ORGANIZATION_BLOCK MAIN:OB1
TITLE= ==========================================
//  初始化与急停复位
//  ==========================================
BEGIN
Network 1 //  首次扫描初始化（清零状态与输出）
LD     SM0.1  // 读取 首次扫描(SM0.1)
MOVB   0, VB100  // 开机顺控状态清零
MOVB   0, VB101  // 关机顺控状态清零
R      Q0.0, 8  // 复位输出 Q0.0~Q0.7
R      Q1.0, 1  // 复位 直流电源(Q1.0)，数量=1
R      M0.0, 2  // 复位 M0.0~M0.1（泵使能）

Network 2 //  急停处理（I0.3）
LD     I0.3  // 读取 急停(I0.3)
MOVB   0, VB100  // 开机顺控状态清零
MOVB   0, VB101  // 关机顺控状态清零
R      Q0.0, 8  // 复位输出 Q0.0~Q0.7
R      Q1.0, 1  // 复位 直流电源(Q1.0)，数量=1
R      M0.0, 2  // 复位 M0.0~M0.1（泵使能）

// ==========================================
// 开机关机触发
// ==========================================
Network 3 //  开机触发（I0.1）
LD     I0.1  // 读取 开机按钮(I0.1)
AN     I0.3  // 与非 急停(I0.3)
AB=    VB100, 0  // 判断 开机顺控状态(VB100) = 0
AB=    VB101, 0  // 判断 关机顺控状态(VB101) = 0
MOVB   10, VB100  // 开机进入步骤10（补水）

Network 4 //  关机触发（I0.2）
LD     I0.2  // 读取 关机按钮(I0.2)
AN     I0.3  // 与非 急停(I0.3)
MOVB   0, VB100  // 开机顺控状态清零
MOVB   10, VB101  // 关机进入步骤10（立即停）

// ==========================================
// AE08 模拟量采集 (8路 4-20mA)
// 说明：按 S7-200 SMART 的固定映射惯例，首个右侧信号模块的模拟量起始通常为 AIW16。
// 若你的系统块里显示的起始地址不同，只需改这里的 AIWxx。
// ==========================================
Network 5 //  AE08 CH0 采集：压力 -> VW1000
LD     SM0.0  // 读取 Always_On(SM0.0)
MOVW   AIW16, VW1000  // 采集模拟量到 压力原始值(VW1000)

Network 6 //  AE08 CH1 采集：阳极液位 -> VW1002
LD     SM0.0  // 读取 Always_On(SM0.0)
MOVW   AIW18, VW1002  // 采集模拟量到 阳极液位原始值(VW1002)

Network 7 //  AE08 CH2 采集：阴极液位 -> VW1004
LD     SM0.0  // 读取 Always_On(SM0.0)
MOVW   AIW20, VW1004  // 采集模拟量到 阴极液位原始值(VW1004)

Network 8 //  AE08 CH3 预留 -> VW1010
LD     SM0.0  // 读取 Always_On(SM0.0)
MOVW   AIW22, VW1010  // 采集模拟量到 VW1010

Network 9 //  AE08 CH4 预留 -> VW1012
LD     SM0.0  // 读取 Always_On(SM0.0)
MOVW   AIW24, VW1012  // 采集模拟量到 VW1012

Network 10 //  AE08 CH5 预留 -> VW1014
LD     SM0.0  // 读取 Always_On(SM0.0)
MOVW   AIW26, VW1014  // 采集模拟量到 VW1014

Network 11 //  AE08 CH6 预留 -> VW1016
LD     SM0.0  // 读取 Always_On(SM0.0)
MOVW   AIW28, VW1016  // 采集模拟量到 VW1016

Network 12 //  AE08 CH7 预留 -> VW1018
LD     SM0.0  // 读取 Always_On(SM0.0)
MOVW   AIW30, VW1018  // 采集模拟量到 VW1018

// ==========================================
// 开机顺控状态机 (VB100)
// ==========================================
Network 13 //  开机步骤10：开制水+开补水阀
LD     SM0.0  // 读取 Always_On(SM0.0)
AB=    VB100, 10  // 判断 开机顺控状态(VB100) = 10
S      Q0.7, 1  // 置位 制水机(Q0.7)
S      Q0.2, 1  // 置位 阳极补水阀(Q0.2)
S      Q0.3, 1  // 置位 阴极补水阀(Q0.3)

Network 14 //  开机步骤10：阳极液位达标关阳极补水
LD     SM0.0  // 读取 Always_On(SM0.0)
AB=    VB100, 10  // 判断 开机顺控状态(VB100) = 10
AW>=   VW1002, 100  // 模拟量阈值比较（达到则进入下一步）
R      Q0.2, 1  // 复位 阳极补水阀(Q0.2)，数量=1

Network 15 //  开机步骤10：阴极液位达标关阴极补水
LD     SM0.0  // 读取 Always_On(SM0.0)
AB=    VB100, 10  // 判断 开机顺控状态(VB100) = 10
AW>=   VW1004, 100  // 模拟量阈值比较（达到则进入下一步）
R      Q0.3, 1  // 复位 阴极补水阀(Q0.3)，数量=1

Network 16 //  开机步骤10：两路补水阀都关 -> 进入步骤20
LD     SM0.0  // 读取 Always_On(SM0.0)
AB=    VB100, 10  // 判断 开机顺控状态(VB100) = 10
AN     Q0.2  // 与非 阳极补水阀(Q0.2)
AN     Q0.3  // 与非 阴极补水阀(Q0.3)
MOVB   20, VB100  // 开机进入步骤20（空压机）

Network 17 //  开机步骤20：启动空压机并计时3秒
LD     SM0.0  // 读取 Always_On(SM0.0)
AB=    VB100, 20  // 判断 开机顺控状态(VB100) = 20
S      Q0.6, 1  // 置位 空压机(Q0.6)
TON    T37, 30  // 定时器 T37：3秒（100ms基准）

Network 18 //  开机步骤20：3秒到 -> 进入步骤30
LD     SM0.0  // 读取 Always_On(SM0.0)
AB=    VB100, 20  // 判断 开机顺控状态(VB100) = 20
A      T37  // 与 3秒延时(T37)
MOVB   30, VB100  // 开机进入步骤30（阳极阀）

Network 19 //  开机步骤30：开阳极电磁阀并计时3秒
LD     SM0.0  // 读取 Always_On(SM0.0)
AB=    VB100, 30  // 判断 开机顺控状态(VB100) = 30
S      Q0.4, 1  // 置位 阳极电磁阀(Q0.4)
TON    T38, 30  // 定时器 T38：3秒（100ms基准）

Network 20 //  开机步骤30：3秒到 -> 进入步骤40
LD     SM0.0  // 读取 Always_On(SM0.0)
AB=    VB100, 30  // 判断 开机顺控状态(VB100) = 30
A      T38  // 与 3秒延时(T38)
MOVB   40, VB100  // 开机进入步骤40（阳极泵）

Network 21 //  开机步骤40：启动阳极泵（使能位）
LD     SM0.0  // 读取 Always_On(SM0.0)
AB=    VB100, 40  // 判断 开机顺控状态(VB100) = 40
S      M0.0, 1  // 置位 阳极泵使能(M0.0)

Network 22 //  开机步骤40：压力达标 -> 进入步骤50
LD     SM0.0  // 读取 Always_On(SM0.0)
AB=    VB100, 40  // 判断 开机顺控状态(VB100) = 40
AW>=   VW1000, 1000  // 模拟量阈值比较（达到则进入下一步）
MOVB   50, VB100  // 开机进入步骤50（阴极泵）

Network 23 //  开机步骤50：启动阴极泵（使能位）并计时3秒
LD     SM0.0  // 读取 Always_On(SM0.0)
AB=    VB100, 50  // 判断 开机顺控状态(VB100) = 50
S      M0.1, 1  // 置位 阴极泵使能(M0.1)
TON    T39, 30  // 定时器 T39：3秒（100ms基准）

Network 24 //  开机步骤50：3秒到 -> 进入步骤60
LD     SM0.0  // 读取 Always_On(SM0.0)
AB=    VB100, 50  // 判断 开机顺控状态(VB100) = 50
A      T39  // 与 3秒延时(T39)
MOVB   60, VB100  // 开机进入步骤60（阴极阀）

Network 25 //  开机步骤60：开阴极液体阀并计时5分钟
LD     SM0.0  // 读取 Always_On(SM0.0)
AB=    VB100, 60  // 判断 开机顺控状态(VB100) = 60
S      Q0.5, 1  // 置位 阴极液体阀(Q0.5)
TON    T40, 3000  // 定时器 T40：5分钟（100ms基准）

Network 26 //  开机步骤60：5分钟到 -> 进入步骤70
LD     SM0.0  // 读取 Always_On(SM0.0)
AB=    VB100, 60  // 判断 开机顺控状态(VB100) = 60
A      T40  // 与 5分钟延时(T40)
MOVB   70, VB100  // 开机进入步骤70（直流电源）

Network 27 //  开机步骤70：使能直流电源 -> 运行状态
LD     SM0.0  // 读取 Always_On(SM0.0)
AB=    VB100, 70  // 判断 开机顺控状态(VB100) = 70
S      Q1.0, 1  // 置位 直流电源(Q1.0)
MOVB   100, VB100  // 开机完成：运行状态

// ==========================================
// 关机顺控状态机 (VB101)
// ==========================================
Network 28 //  关机步骤10：立即关闭阀/泵/制水/直流电源
LD     SM0.0  // 读取 Always_On(SM0.0)
AB=    VB101, 10  // 判断 关机顺控状态(VB101) = 10
R      Q1.0, 1  // 复位 直流电源(Q1.0)，数量=1
R      Q0.2, 2  // 复位 阳极补水阀(Q0.2)，数量=2
R      Q0.7, 1  // 复位 制水机(Q0.7)，数量=1
R      M0.1, 1  // 复位 阴极泵使能(M0.1)，数量=1
R      Q0.5, 1  // 复位 阴极液体阀(Q0.5)，数量=1
R      M0.0, 1  // 复位 阳极泵使能(M0.0)，数量=1
R      Q0.4, 1  // 复位 阳极电磁阀(Q0.4)，数量=1
MOVB   20, VB101  // 关机进入步骤20（延时）

Network 29 //  关机步骤20：延时30分钟
LD     SM0.0  // 读取 Always_On(SM0.0)
AB=    VB101, 20  // 判断 关机顺控状态(VB101) = 20
TON    T41, 18000  // 定时器 T41：30分钟（100ms基准）

Network 30 //  PWM向导调用（如未使用PWM可忽略）
LD     SM0.0  // 读取 Always_On(SM0.0)
=      L60.0  // 写入 临时位(Always_On缓存)(L60.0)
LDN    M0.0  // 读取(取反) 阳极泵使能(M0.0)
=      L63.7  // 写入 临时位(PWM_RUN)(L63.7)
LD     L60.0  // 读取 临时位(Always_On缓存)(L60.0)
CALL   SBR0, L63.7, 20, 10, VB100  // 调用 PWM0_RUN：RUN/Cycle/Pulse/Error
Network 31 //  默认输出：AQW32=5V（测试）
// 配置默认5V输出测试
LD     SM0.0  // 读取 Always_On(SM0.0)
MOVW   13824, AQW32  // 输出 AO0(阳极泵给定)：默认 5V（测试）
END_ORGANIZATION_BLOCK
SUBROUTINE_BLOCK PWM0_RUN:SBR0
TITLE=该指令由 PTO/PWM 向导生成，旨在与输出 Q0.0 配合使用. 该输出用作采用同步更新并基于 毫秒 时基的 PWM.
VAR_INPUT
RUN:BOOL;	// 运行/停止
Cycle:WORD;	// 周期时间 (2-65535 ms)
Pulse:WORD;	// 脉冲时间宽度 (0-65535)
END_VAR
VAR_OUTPUT
Error:BYTE;
END_VAR
VAR
Control_Byte:BYTE;
Tmp_Array:BYTE;
Tmp_Array2:BYTE;
Tmp_Array3:BYTE;
Tmp_Array4:BYTE;
Tmp_Array5:BYTE;
END_VAR
BEGIN
Network 1 //  首次扫描初始化（清零状态与输出）

END_SUBROUTINE_BLOCK

